(* IEC 61131-3 sources: POMIRTS_lab3/AS/Library_2/net2000, 3 files *)

(* ---- net2000.typ ---- *)
TYPE
	NET2PV : STRUCT
		PvLength	: UINT ;
		PvName	: ARRAY[0..31] OF SINT ;
	END_STRUCT;
	NET2EVT : STRUCT
		nvars	: UINT ;
	END_STRUCT;
	NET2CAN : STRUCT
		nnodes	: USINT ;
		basis	: UINT ;
	END_STRUCT;
	NET2CONFIGURATION : STRUCT
		station	: USINT ;
		task_class	: SINT ;
		retry	: USINT ;
		master	: USINT ;
		device	: UDINT ;
		mode	: UDINT ;
		ixtabsize	: UINT ;
		t_response	: UINT ;
		t_cross	: UINT ;
		l7length	: UDINT ;
		status	: UINT ;
		reset	: USINT ;
		freeze	: USINT ;
		close	: USINT ;
		CAN	: NET2CAN ;
		EVT	: NET2EVT ;
	END_STRUCT;
END_TYPE

(* ---- net2000.fun ---- *)
{REDUND_ERROR} FUNCTION_BLOCK NET2write (* NET2000 - Write-FUB *)
	VAR_INPUT
		enable	:BOOL;
		destadr	:DINT;
		pvlist	:UDINT;
		pvnum	:UINT;
		dataarea	:UDINT;
		datlng	:UINT;
	END_VAR
	VAR_OUTPUT
		ok	:BOOL;
		status	:UINT;
		record	:UDINT;
		reqcnt	:UDINT;
		rqdatlng	:UINT;
	END_VAR
	VAR
		InternalData	:STRING[175];
	END_VAR
END_FUNCTION_BLOCK
{REDUND_ERROR} FUNCTION_BLOCK NET2read (* NET2000 - Read-FUB *)
	VAR_INPUT
		enable	:BOOL;
		destadr	:DINT;
		pvlist	:UDINT;
		pvnum	:UINT;
		dataarea	:UDINT;
		datlng	:UINT;
	END_VAR
	VAR_OUTPUT
		ok	:BOOL;
		status	:UINT;
		record	:UDINT;
		reqcnt	:UDINT;
		rqdatlng	:UINT;
	END_VAR
	VAR
		InternalData	:STRING[175];
	END_VAR
END_FUNCTION_BLOCK

(* ---- net2000.var ---- *)
VAR CONSTANT

END_VAR
